// TIA Portal V20 export
DATA_BLOCK "Oil_DB"   // DB40
// stored: InstanceOfName Oil, InstanceOfType FB
"Oil"
   // VAR_INPUT
   //    Safety_OK : Bool;
   //    Pump_status : Bool;
   //    Pump_error : Bool;
   //    Pallette_Moving : Bool;
   // END_VAR
   // VAR_OUTPUT
   //    Pump : Bool;
   //    Main_Valve : Bool;
   //    Preparation_Valve : Bool;
   //    Nozzle_Valve : Bool;
   //    Pump_Volume_Output : Int;
   // END_VAR
   // VAR
   //    Pump_Reset { S7_SetPoint := 'True'} : TON_TIME;
   //    Pump_Volume { S7_SetPoint := 'True'} : Real;
   //    Oil_Station_Enable : Bool;
   // END_VAR
BEGIN
END_DATA_BLOCK
